PROGRAM EventLogger
VAR
	bInit:			BOOL:=TRUE;
	
	aAlarm:			ARRAY[0..Parameter.cAnzEvents] OF FB_Event;
	aMessage:		ARRAY[0..Parameter.cAnzEvents] OF FB_Event;
	aWarnung:		ARRAY[0..Parameter.cAnzEvents] OF FB_Event;
	aErrorLog:		ARRAY[0..Parameter.cAnzEvents] OF FB_Event;
	
	i:				INT;
	j:				INT;
	
	
	
	fbTime 			: NT_GetTime;
END_VAR
VAR PERSISTENT	
	aLoggedEvents:	ARRAY[0..Parameter.cAnzLoggedEvents] OF ST_EventTabelle;
END_VAR

IF bInit THEN
    bInit := FALSE; 
	//Station 1
	aAlarm[13].setText('error', 'Aktor 1 hat Arbeitsposition nicht erreicht oder verloren');
	aAlarm[14].setText('error', 'Aktor 1 hat Ruheposition nicht erreicht oder verloren');
	aAlarm[15].setText('error', 'Aktor 2 hat Arbeitsposition nicht erreicht oder verloren');
	aAlarm[16].setText('error', 'Aktor 2 hat Ruheposition nicht erreicht oder verloren');
	aAlarm[17].setText('error', 'Aktor 3 hat Arbeitsposition nicht erreicht oder verloren');
	aAlarm[18].setText('error', 'Aktor 3 hat Ruheposition nicht erreicht oder verloren');
	aAlarm[19].setText('error', 'Aktor 4 hat Arbeitsposition nicht erreicht oder verloren');
	aAlarm[20].setText('error', 'Aktor 4 hat Ruheposition nicht erreicht oder verloren');
	aAlarm[21].setText('error', 'Aktor 5 hat Arbeitsposition nicht erreicht oder verloren');
	aAlarm[22].setText('error', 'Aktor 5 hat Ruheposition nicht erreicht oder verloren');
	aAlarm[23].setText('error', 'Aktor 6 hat Arbeitsposition nicht erreicht oder verloren');
	aAlarm[24].setText('error', 'Aktor 6 hat Ruheposition nicht erreicht oder verloren');
	
	aAlarm[39].setText('error', 'Kein Teil in Aufnahme. Station per Reset zurücksetzen');
	aAlarm[40].setText('error', 'Not-Halt muss getestet werden');
	

	//	
	aAlarm[100].setText('error', 'Fehler Safety. Anlage mittels Hauptschalter neu starten');
	
	aAlarm[253].setText('error', 'Es wurde {0} Mal in Folge Ausschuss erkannt. Bitte Fehler beheben und "Stoerung Quittieren" betaetigen');
	aAlarm[257].setText('error', 'Luftdruck ist ausserhalb von 5.0 - 6.0bar');
	//
	
	aAlarm[262].setText('error', 'Informationen konnten nicht an Datenbank gesendet werden. Um erneut zu senden, Störung quittieren');
	aAlarm[264].setText('error', 'Senden an Datenbank nicht möglich. (Queue voll) Bitte an Support wenden');

	//
	aErrorLog[230].setText('error', 'Anlage kann nicht gestartet werden, da der Programmablaufunterbruch aktiv ist');
	aErrorLog[231].setText('error', 'Anlage kann nicht gestartet werden, da sich ein Aktor in der falschen Position befindet (im Handbetrieb verfahren)');
	aErrorLog[232].setText('error', 'Anlage kann nicht gestartet werden, da der Handbetrieb aktiviert ist');
	aErrorLog[233].setText('error', 'Anlage kann nicht gestartet werden, da sie nicht fertig Initialisiert ist');
	aErrorLog[234].setText('error', 'Anlage kann nicht gestartet werden, da kein Artikel vorgewaehlt wurde');
	aErrorLog[235].setText('error', 'Anlage kann nicht gestartet werden, da zu viel Ausschuss in Folge produziert wurde');
	aErrorLog[250].setText('error', '{0} sollte sich in der {1} befinden (Falsche Position beim verlassen des Handbetriebs)');
	//
	aErrorLog[260].setText('error', 'Überstromschutzklemme {0} Kanal {1} {2}');
	aErrorLog[261].setText('error', 'MQTT-Message Timeout. Art: {0}, Kennung: {1}');
	aErrorLog[263].setText('error', 'MQTT-Message Error. Art: {0}, Grund: {1}, Kennung: {2}');
	//
	//
	aErrorLog[300].setText('error', '{0}');
	//
	aWarnung[300].setText('warnung', '{0}');
	//
	aMessage[10].setText('info', 'Init wartet auf {0}');
	aMessage[11].setText('info', 'Init fertig');
	aMessage[300].setText('info', '{0}');
	
	
	FOR i := 0 TO Parameter.cAnzLoggedEvents DO
		IF			aLoggedEvents[i].sStatus = 'Aktiv'
			or		aLoggedEvents[i].bPinned THEN
			aLoggedEvents[i].sStatus := 'Cleared';
			aLoggedEvents[i].bPinned := FALSE;
		END_IF
	END_FOR
END_IF

fbTime(START := TRUE);
fbTime(START := FALSE);

FOR i := 0 TO Parameter.cAnzEvents DO
	aAlarm[i](nID := i);
	aMessage[i](nID := i);
	aWarnung[i](nID := i);
	aErrorLog[i](nID := i);
END_FOR

METHOD logEvent
VAR_INPUT
	nEventId:	INT;
	sText:		STRING(255);
	sSeverity: 	STRING;
	bPin:		BOOL;
END_VAR
VAR
	i:			INT;
END_VAR
FOR i := Parameter.cAnzLoggedEvents-1 TO 0 BY -1 DO
	
	IF 		NOT aLoggedEvents[i].bPinned 		//Nicht gepinnte Events schieben
		OR		bPin THEN						//Gepinnte Events auch schieben falls der neue gepinnt werden soll
		aLoggedEvents[i+1] := aLoggedEvents[i];
	ELSE					
		EXIT;
	END_IF
END_FOR



aLoggedEvents[i+1].bPinned := bPin;
aLoggedEvents[i+1].sText := sText;
aLoggedEvents[i+1].sSeverity := sSeverity;
aLoggedEvents[i+1].nEventId := nEventId;
aLoggedEvents[i+1].sTimestamp := SYSTEMTIME_TO_STRING(fbTime.TIMESTR);

IF			bPin THEN
	aLoggedEvents[i+1].sStatus := 'Aktiv';
ELSE 
	aLoggedEvents[i+1].sStatus := '';
END_IF
END_METHOD

METHOD unpinEvent
VAR_INPUT
	nID:		INT;
END_VAR
FOR i := 0 TO Parameter.cAnzLoggedEvents DO	
	IF 			(aLoggedEvents[i].nEventId = nID)
		AND	 	aLoggedEvents[i].bPinned THEN
		aLoggedEvents[i].sStatus := 'Cleared';
		aLoggedEvents[i].bPinned := FALSE;
	END_IF
END_FOR
END_METHOD

END_PROGRAM

(* stored: Version 1.1.0.1, ProductVersion 3.1.4024.12
   POU EventLogger: Id {1500f798-262a-440f-8446-1df31fe2b41e}, SpecialFunc None
   Method logEvent: Id {dddbf2d9-2d14-4a05-8ba4-3074f981098c}
   Method unpinEvent: Id {9363361b-7b0a-4201-937b-a77ae2c26f1c} *)
